Staubli VAL3: sad_project_1.pjx

--- sad_project_1.pjx ---
Parameters version=s7.7.1 stackSize=5000 millimeterUnit=true
Program file=check_cmt.pgx
Program file=motion_cntl.pgx
Program file=open_socket.pgx
Program file=read_data.pgx
Program file=send_data.pgx
Program file=show_data.pgx
Program file=start.pgx
Program file=stop.pgx
Data file=sad_project_1.dtx

--- sad_project_1.dtx ---
sio sioASCII = {link=Socket\trsf_sv}
public bool check_status
public num Ref_Vel
public mdesc mNomSpeed = {tmax=100, rmax=100, leave=0.1, reach=0.1, blend=off}
public jointRx Jnt_cnfg = {j3=90, j5=90, j6=90}
public tool tTool = {z=200, fatherId=flange[0], ioLink=valve1}
public mdesc cnst_vel = {tmax=100, rmax=100, leave=0.1, reach=0.1, blend=cartesian}
public frame fReference = {x=1365.054, y=-125.975, z=-500, fatherId=world[0]}
public pointRx Pnt_1st_lyr[2]
  [0] = {y=-1000, rx=-180, rz=-90, shoulder=lefty, elbow=epositive, wrist=wpositive, fatherId=fReference[0]}
  [1] = {y=1000, rx=-180, rz=-90, shoulder=lefty, elbow=epositive, wrist=wpositive, fatherId=fReference[0]}
public pointRx Pnt_2nd_lyr[4]
  [0] = {y=1000, z=77, rx=180, rz=-90, shoulder=lefty, elbow=epositive, wrist=wpositive, fatherId=fReference[0]}
  [1] = {y=-1000, z=77, rx=180, rz=-90, shoulder=lefty, elbow=epositive, wrist=wpositive, fatherId=fReference[0]}
  [2] = {y=-1000, z=22, rx=180, rz=-90, shoulder=lefty, elbow=epositive, wrist=wpositive, fatherId=fReference[0]}
  [3] = {y=1000, z=22, rx=180, rz=-90, shoulder=lefty, elbow=epositive, wrist=wpositive, fatherId=fReference[0]}
public pointRx Pnt_3rd_lyr[4]
  [0] = {y=1000, z=99, rx=180, rz=-90, shoulder=lefty, elbow=epositive, wrist=wpositive, fatherId=fReference[0]}
  [1] = {y=-1000, z=99, rx=180, rz=-90, shoulder=lefty, elbow=epositive, wrist=wpositive, fatherId=fReference[0]}
  [2] = {y=-1000, z=44, rx=180, rz=-90, shoulder=lefty, elbow=epositive, wrist=wpositive, fatherId=fReference[0]}
  [3] = {y=1000, z=44, rx=180, rz=-90, shoulder=lefty, elbow=epositive, wrist=wpositive, fatherId=fReference[0]}
public pointRx Pnt_4th_lyr[4]
  [0] = {y=1000, z=116, rx=180, rz=-90, shoulder=lefty, elbow=epositive, wrist=wpositive, fatherId=fReference[0]}
  [1] = {y=-1000, z=116, rx=180, rz=-90, shoulder=lefty, elbow=epositive, wrist=wpositive, fatherId=fReference[0]}
  [2] = {y=-1000, z=66, rx=180, rz=-90, shoulder=lefty, elbow=epositive, wrist=wpositive, fatherId=fReference[0]}
  [3] = {y=1000, z=66, rx=180, rz=-90, shoulder=lefty, elbow=epositive, wrist=wpositive, fatherId=fReference[0]}
public trsf trTrsf
public bool spd_cntl

--- start.pgx ---
program start()
begin
  disablePower()
  cls()
  userPage()
  title(" Concrete 3D Printer ")
  putln("Written by Erfan.")
  setProfile("Manual","123")
  if getProfile() == "Manual"
    putln("Profile is set to Remote Control.")
  endIf
  delay(3)
  enablePower()
  if(watch(isPowered(),3) == false)
    putln("Arm power supply cannot be swithced on.")
  endIf
  putln("Arm power is now switched on.")
  delay(5)
  taskCreate "SocketOpening",10,open_socket()
  taskCreate "CheckComnunic",20,check_cmt()
  wait(check_status == true)
  delay(2)
  taskCreate "DataReading",40,read_data()
  taskCreate "MotionControl",40,motion_cntl()
  taskCreate "DataDisplay",40,show_data()
  taskCreate "DataSending",50,send_data()

  //////////////////////////////////////////
  // Go to configuration
  spd_cntl = false
  resetMotion()
  setMonitorSpeed(100)
  movej(Jnt_cnfg[0],tTool[0],cnst_vel[0])
  waitEndMove()

  // Go to Start point - 1st Layer
  spd_cntl = false
  setMonitorSpeed(100)
  movel(Pnt_1st_lyr[0],tTool[0],mNomSpeed[0])
  waitEndMove()

  // Printing - 1st Layer
  setProfile("Automatic","123")
  spd_cntl = true
  resetMotion()
  movel(Pnt_1st_lyr[1],tTool[0],mNomSpeed[0])
  waitEndMove()


  resetMotion()
  setProfile("Manual","123")
  // Go to Start point - 2nd Layer
  spd_cntl = false
  resetMotion()
  setMonitorSpeed(100)
  movel(Pnt_2nd_lyr[0],tTool[0],cnst_vel[0])
  waitEndMove()
  movel(Pnt_2nd_lyr[1],tTool[0],cnst_vel[0])
  waitEndMove()
  movel(Pnt_2nd_lyr[2],tTool[0],cnst_vel[0])
  waitEndMove()

  // Printing - 2nd Layer
  setProfile("Automatic","123")
  spd_cntl = true
  resetMotion()
  movel(Pnt_2nd_lyr[3],tTool[0],mNomSpeed[0])
  waitEndMove()

  // Go to Start point - 3rd Layer
  setProfile("Manual","123")
  spd_cntl = false
  resetMotion()
  setMonitorSpeed(100)
  movel(Pnt_3rd_lyr[0],tTool[0],cnst_vel[0])
  waitEndMove()
  movel(Pnt_3rd_lyr[1],tTool[0],cnst_vel[0])
  waitEndMove()
  movel(Pnt_3rd_lyr[2],tTool[0],cnst_vel[0])
  waitEndMove()

  // Printing - 3rd Layer
  setProfile("Automatic","123")
  spd_cntl = true
  resetMotion()
  movel(Pnt_3rd_lyr[3],tTool[0],mNomSpeed[0])
  waitEndMove()


  // Go to Start point - 4th Layer
  setProfile("Manual","123")
  spd_cntl = false
  resetMotion()
  setMonitorSpeed(100)
  movel(Pnt_4th_lyr[0],tTool[0],cnst_vel[0])
  waitEndMove()
  movel(Pnt_4th_lyr[1],tTool[0],cnst_vel[0])
  waitEndMove()
  movel(Pnt_4th_lyr[2],tTool[0],cnst_vel[0])
  waitEndMove()


  // Printing - 4th Layer
  setProfile("Automatic","123")
  spd_cntl = true
  resetMotion()
  movel(Pnt_4th_lyr[3],tTool[0],mNomSpeed[0])
  waitEndMove()

  // Go to configuration
  spd_cntl = false
  resetMotion()
  setMonitorSpeed(100)
  movej(Jnt_cnfg[0],tTool[0],cnst_vel[0])
  waitEndMove()

  stopMove()
  disablePower()


  ///////////////////////////////////////////


end

--- motion_cntl.pgx ---
public program motion_cntl()
begin

  do

    wait(spd_cntl == true)
    setMonitorSpeed(Ref_Vel)

  until check_status != true

end

--- open_socket.pgx ---
public program open_socket()
begin

  sioCtrl(sioASCII,"port",11002)
  //sioCtrl(sioASCII,"port",1002)
  //sioCtrl(sioASCII,"target","10.3.1.185")
  //sioCtrl(sioASCII,"target","10.10.5.1")
  sioCtrl(sioASCII,"target","169.254.209.1")
  sioCtrl(sioASCII,"timeout",10)
  sioCtrl(sioASCII,"endOfString",13)
  sioCtrl(sioASCII,"nangle",true)

  putln("The communication socket is open.")

  check_status = false

end

--- read_data.pgx ---
public program read_data()
  local string sInputData_1
  local num nRec
  local num nReceived
  local num nInputData_1
begin

  putln("Start to read data !")

  do
    sInputData_1 = ""
    do
      nReceived=sioGet(sioASCII,nRec)
      sInputData_1 = sInputData_1 + chr(nRec)

    until nRec == 13 or nReceived == -1

    if nReceived != 1
      check_status = false
      stopMove()
      cls()
      putln("Communication error !")
      enablePower()
    endIf

    toNum(sInputData_1 , nInputData_1, check_status)

    //put("Reference Velocity [mm/s]: ")
    //put(nInputData_1)
    //putln("")
    Ref_Vel = nInputData_1

   // putln(Ref_Vel)


  // delay(0.001)

  until check_status != true

end

--- send_data.pgx ---
program send_data()
  local string snd_msg
  local num i
  local num nSent
begin

  putln("Start to send data !")

  do

  snd_msg = toString(".4",getSpeed(tTool)) + chr(13) + chr(10)

  for i=0 to len(snd_msg)-1
    nSent = sioSet(sioASCII,asc(snd_msg,i))

    if nSent != 1
      check_status = false
      stopMove()
      cls()
      putln("Communication error !")
      disablePower()
    endIf


  endFor

  //putln(snd_msg)

  //cls()
  delay(.4)

  until check_status != true


end

--- show_data.pgx ---
public program show_data()
begin

   do
    cls()
    put("Reference Velocity [mm/s]: ")
    put(Ref_Vel)
    putln("")
    //cls()
    put("Robot Velocity [mm/s]: ")
    put(getSpeed(tTool))
    putln("")
    //cls()
    put("Error (Ref-Rob) [mm/s]: ")
    put(Ref_Vel - getSpeed(tTool))
    putln("")
    //cls()
    put("Current position: ")
    put(getMoveId())
    putln("")


    delay(0.001)
    //putln("")
  until check_status != true

end
